{attribute 'qualified_only'}
//{attribute 'strict'}
TYPE ConveyorMode :
(
	IDLE,
	FORWARD,
	BACKWARD,
	STOP,
	
	size
);
END_TYPE

(* stored: Version 1.1.0.1, ProductVersion 3.1.4024.11
   DUT ConveyorMode: Id {cf678971-d1f4-4b67-8437-64e465d0ac0b} *)
